// TIA Portal V17 export
// export: Created 2025-03-07T09:17:49.798012Z, ExportSetting WithDefaults, DisplayName Totally Integrated Automation Portal, DisplayVersion V17 Update 8, DisplayName TIA Portal Openness, DisplayVersion V17 Update 8, DisplayName TIA Portal Version Control Interface, DisplayVersion V17, DisplayName SINAMICS Startdrive Advanced, DisplayVersion V17 SP2, DisplayName SINAMICS Startdrive G110M, G120, G120C, G120D, G120P, G115D, DisplayVersion V17 SP2, DisplayName SINAMICS Startdrive G130, G150, S120, S150, SINAMICS MV, S210, DisplayVersion V17 SP2, DisplayName STEP 7 Professional, DisplayVersion V17 Update 8, DisplayName SINUMERIK ONE STEP 7 Toolbox, DisplayVersion V17 Update 12, DisplayName SINUMERIK 840D sl STEP 7 Toolbox, DisplayVersion V17 Update 12, DisplayName STEP 7 Safety, DisplayVersion V17 Update 6, DisplayName WinCC Advanced, DisplayVersion V17 Update 8
DATA_BLOCK "DB2122_HT10"   // DB2122
{ S7_Optimized_Access := 'FALSE'; DB_Accessible_From_OPC_UA := 'FALSE' }
AUTHOR : ETXETAR
VERSION : 1.0
// stored: AutoNumber false, DBAccessibleFromOPCUA false, DBAccessibleFromWebserver true, IsOnlyStoredInLoadMemory false, IsWriteProtectedInAS false
   VAR
      INPUT_HT10_EMERGENCY_STOP : Bool;   // INPUT HT8 EMERGENCY STOP / INPUT HT10 EMERGENCY STOP
      HT10_EMERGENCY_STOP_ACTIVE : Bool;   // HT8 EMERGENCY STOP ACTIVE / HT10 EMERGENCY STOP ACTIVE
      INPUTS : "HT10_INPUTS";   // HT10 INPUTS
      ENABLE_CHANGE { S7_SetPoint := 'True'} : "HT10_ENABLE_CHANGE";
   END_VAR
BEGIN
END_DATA_BLOCK
